FUNCTION_BLOCK FB_WhiteSpaces
VAR_INPUT
END_VAR
VAR_OUTPUT
	sWhiteSpace : T_MaxString;
END_VAR
VAR
	bInit : BOOL;
	i : UINT;

END_VAR

IF NOT bInit THEN
	bInit := TRUE;
	FOR i := 1 TO SIZEOF(T_MAXSTRING) DO
		sWhiteSpace := Concat(sWhiteSpace,' ');
	END_FOR
END_IF

END_FUNCTION_BLOCK

(* stored: Version 1.1.0.1, ProductVersion 3.1.4022.16
   POU FB_WhiteSpaces: Id {9cb5ef31-20f8-45bc-84eb-aecd12ded6a1}, SpecialFunc None *)
